FUNCTION_BLOCK "G020M_Code"
TITLE =G020G CCOMPRESSED AIR PRESSURE STEEP 21 - 24
//COPYRIGHT:    (C) 2009  BUHLER AG, CH-9240 UZWIL, SWITZERLAND
//
//PRODUCT:      WinCoS_BIW01_09
//
//TITLE:        CCOMPRESSED AIR PRESSURE STEEP 21 - 24
//                General group control
//                Allgemeine Gruppensteuerung
//
//--------------------------------------------------------------------------------
//
//IDENT:        AUTHOR:             DEPT:                              DATE:
//
//P01_FB120.1.0 K.Renz              CSB41                              29.Sep.2009
//             1st Release
//
//--------------------------------------------------------------------------------
//
//PURPOSE:
//
//MANUAL :
//
//RESTRICTIONS:
//
//--------------------------------------------------------------------------------
AUTHOR : KR
FAMILY : USW
VERSION : 9.9


VAR
  Gr : "GCS7_GrpCtrlSub";	//Standard interface to group
  InOutValue1 : DINT ;	//Data for user
  InOutValue2 : DINT ;	//Data for user
  OutWayConflict : BOOL ;	//Data for user
  OutSelectionOk : BOOL ;	//Data for user
  CmdNewValue : BOOL ;	//Data for user
  CmdNewJob : BOOL ;	//Data for user
  OutCodeOK : BOOL ;	//Data for user
  InEndOfJob : BOOL ;	//Data for user
  staWayOk : BOOL ;	//Data for user
  EdgeStartRelease : BOOL ;	//Data for user
  USW8 : BOOL ;	//Data for user
  USW9 : BOOL ;	//Data for user
  USW10 : BOOL ;	//Data for user
  USW11 : BOOL ;	//Data for user
  USW12 : BOOL ;	//Data for user
  USW13 : BOOL ;	//Data for user
  USW14 : BOOL ;	//Data for user
  USW15 : BOOL ;	//Data for user
  A_1156_MXZ11 : "GCS7_E_Motor";	// Motor
  A_1191_BTE18 : "GCS7_E_AnalogInput"; //Temp sensor
  A_1191_BTE22 : "GCS7_E_AnalogInput"; //Temp sensor

END_VAR
VAR_TEMP
  tmpEnable : BOOL ;
  tmpFlag : BOOL ;
  tmpCmdNext : BOOL ;
  tmpLocal : BOOL ;
  tmpAspOk : BOOL ;
  tmpHWStop : BOOL ;
  tmpInstanzDBNo : INT ;
END_VAR
BEGIN
NETWORK
TITLE =



NETWORK
TITLE =Read command from group control
//Parameter
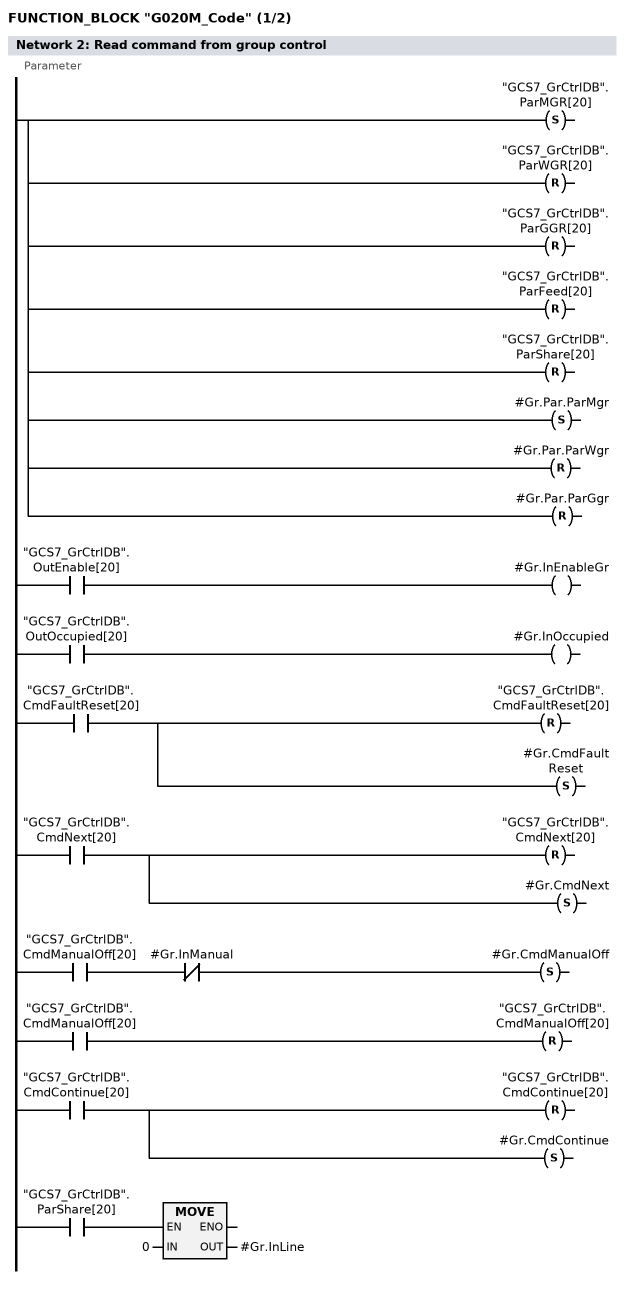
      SET   ;
      S     "GCS7_GrCtrlDB".ParMGR[20];
      R     "GCS7_GrCtrlDB".ParWGR[20];
      R     "GCS7_GrCtrlDB".ParGGR[20];
      R     "GCS7_GrCtrlDB".ParFeed[20];
      R     "GCS7_GrCtrlDB".ParShare[20];
      S     #Gr.Par.ParMgr;
      R     #Gr.Par.ParWgr;
      R     #Gr.Par.ParGgr;
//Command
      A     "GCS7_GrCtrlDB".OutEnable[20];
      =     #Gr.InEnableGr;
      A     "GCS7_GrCtrlDB".OutOccupied[20];
      =     #Gr.InOccupied;
      A     "GCS7_GrCtrlDB".CmdFaultReset[20];
      R     "GCS7_GrCtrlDB".CmdFaultReset[20];
      S     #Gr.CmdFaultReset;
      A     "GCS7_GrCtrlDB".CmdNext[20];
      R     "GCS7_GrCtrlDB".CmdNext[20];
      S     #Gr.CmdNext;
      A     "GCS7_GrCtrlDB".CmdManualOff[20];
      AN    #Gr.InManual;
      S     #Gr.CmdManualOff;
      A     "GCS7_GrCtrlDB".CmdManualOff[20];
      R     "GCS7_GrCtrlDB".CmdManualOff[20];

//      U     "GCS7_GrCtrlDB".CmdManualOff[20]
//      O     "GCS7_GrCtrlDB".OutOccupied[20]
//      R     "GCS7_GrCtrlDB".CmdManualOff[20]
//      S     #Gr.CmdManualOff

      A     "GCS7_GrCtrlDB".CmdContinue[20];
      R     "GCS7_GrCtrlDB".CmdContinue[20];
      S     #Gr.CmdContinue;
//Init Line Number
      A     "GCS7_GrCtrlDB".ParShare[20];
      JCN   WE00;
      L     0;
      T     #Gr.InLine;
WE00: NOP   0;
NETWORK
TITLE =Call Methode Control
// 1. Handle Interface PCControl
// 2. Prepare mode --> ModePassive,ModeActive,ModeIdling
// 3. Reset global flags of the group
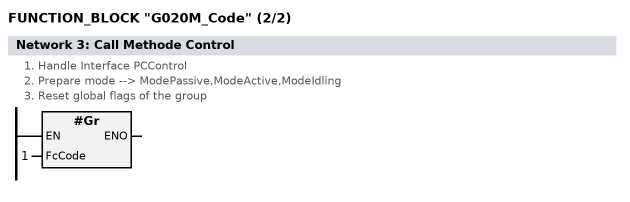
      CALL #Gr (
           FcCode                   := 1);
NETWORK
TITLE =Restart Idling Time

      CLR   ;
      S     #Gr.CmdRestartIdling;
NETWORK
TITLE =Prepare global flags



NETWORK
TITLE =Set Pattern (Target position)



NETWORK
TITLE =Interlocking WayOk



NETWORK
TITLE =Interlocking Autostart

      CLR   ;
      R     #Gr.OutAutostart;
NETWORK
TITLE =Interlocking Enable
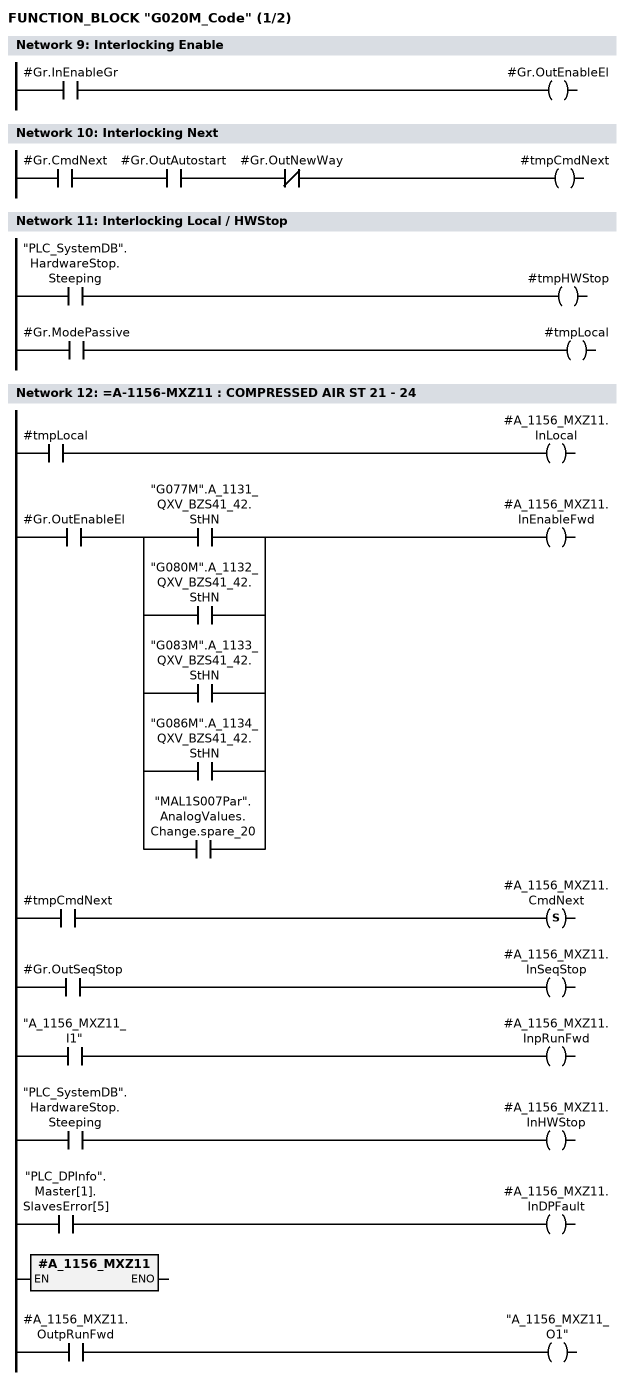

      A     #Gr.InEnableGr;
//      CLR                               // No automatic --> only manual
      =     #Gr.OutEnableEl;

NETWORK
TITLE =Interlocking Next

      A     #Gr.CmdNext;
      A     #Gr.OutAutostart;
      AN    #Gr.OutNewWay;
      =     #tmpCmdNext;

NETWORK
TITLE =Interlocking Local / HWStop

      A     "PLC_SystemDB".HardwareStop.Steeping;
      =     #tmpHWStop;

      A     #Gr.ModePassive;
      =     #tmpLocal;

NETWORK
TITLE ==A-1156-MXZ11 : COMPRESSED AIR ST 21 - 24

      NOP   0;
//-InLocal---
      A     #tmpLocal;
      =     #A_1156_MXZ11.InLocal;
//
//-Interlocking---
      A     #Gr.OutEnableEl;
//=>IS 12.03.2013
      A(    ; //JV190710 =====> min 1 Klappe offen
      O     "G077M".A_1131_QXV_BZS41_42.StHN;
      O     "G080M".A_1132_QXV_BZS41_42.StHN;
      O     "G083M".A_1133_QXV_BZS41_42.StHN;
      O     "G086M".A_1134_QXV_BZS41_42.StHN;
      O     "MAL1S007Par".AnalogValues.Change.spare_20;
      )     ; //JV190710 <======
//<=IS
      =     #A_1156_MXZ11.InEnableFwd;
//
      A     #tmpCmdNext;
      S     #A_1156_MXZ11.CmdNext;
//
      A     #Gr.OutSeqStop;
      =     #A_1156_MXZ11.InSeqStop;
//
//-Read inputs---
      A     "A_1156_MXZ11_I1";
      =     #A_1156_MXZ11.InpRunFwd;
      A     "PLC_SystemDB".HardwareStop.Steeping;
      =     #A_1156_MXZ11.InHWStop;
      A     "PLC_DPInfo".Master[1].SlavesError[5];
      =     #A_1156_MXZ11.InDPFault;
//
//-Set Parameters---
//
//-Call object control---
      CALL #A_1156_MXZ11 ;
//
//-Write outputs---
      A     #A_1156_MXZ11.OutpRunFwd;
      =     "A_1156_MXZ11_O1";
NETWORK
TITLE =Test Fault
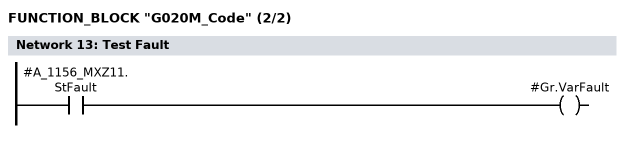

      A     #A_1156_MXZ11.StFault;
      =     #Gr.VarFault;
NETWORK
TITLE =Test Warning

      CLR   ;
      =     #Gr.OutWarning;
NETWORK
TITLE =Test Stopped
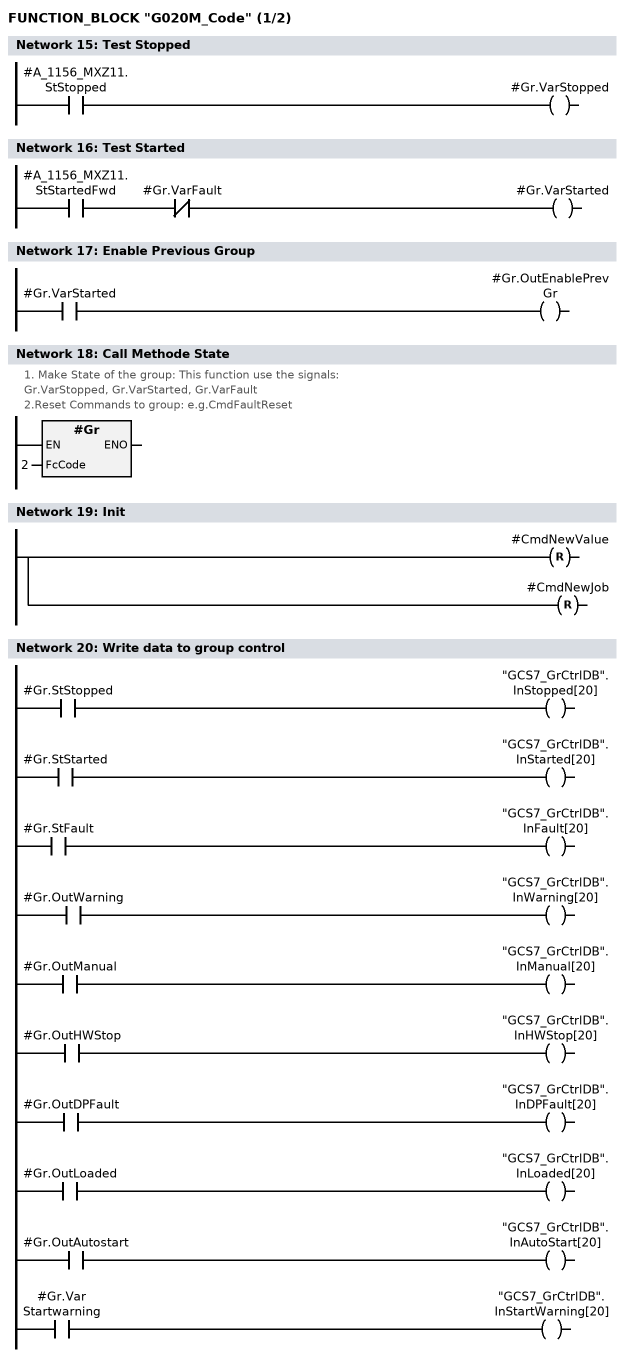

      A     #A_1156_MXZ11.StStopped;
      =     #Gr.VarStopped;
NETWORK
TITLE =Test Started

      A     #A_1156_MXZ11.StStartedFwd;
      AN    #Gr.VarFault;
      =     #Gr.VarStarted;
NETWORK
TITLE =Enable Previous Group

      A     #Gr.VarStarted;
      =     #Gr.OutEnablePrevGr;
NETWORK
TITLE =Call Methode State
//1. Make State of the group: This function use the signals:
//        Gr.VarStopped, Gr.VarStarted, Gr.VarFault
//2.Reset Commands to group: e.g.CmdFaultReset
      CALL #Gr (
           FcCode                   := 2);
NETWORK
TITLE =Init

      SET   ;
      R     #CmdNewValue;
      R     #CmdNewJob;
NETWORK
TITLE =Write data to group control

      A     #Gr.StStopped;
      =     "GCS7_GrCtrlDB".InStopped[20];
      A     #Gr.StStarted;
      =     "GCS7_GrCtrlDB".InStarted[20];
      A     #Gr.StFault;
      =     "GCS7_GrCtrlDB".InFault[20];
      A     #Gr.OutWarning;
      =     "GCS7_GrCtrlDB".InWarning[20];
      A     #Gr.OutManual;
      =     "GCS7_GrCtrlDB".InManual[20];
      A     #Gr.OutHWStop;
      =     "GCS7_GrCtrlDB".InHWStop[20];
      A     #Gr.OutDPFault;
      =     "GCS7_GrCtrlDB".InDPFault[20];
      A     #Gr.OutLoaded;
      =     "GCS7_GrCtrlDB".InLoaded[20];
      A     #Gr.OutAutostart;
      =     "GCS7_GrCtrlDB".InAutoStart[20];
      A     #Gr.VarStartwarning;
      =     "GCS7_GrCtrlDB".InStartWarning[20];
NETWORK
TITLE =End of block
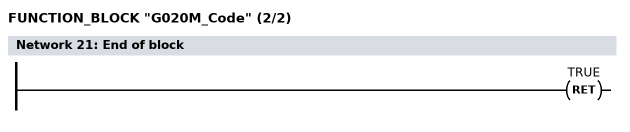

      BE    ;

END_FUNCTION_BLOCK

